// Mitsubishi GX Works2 project: 0924최신화   PLC: Q02U

PROGRAM INPUT
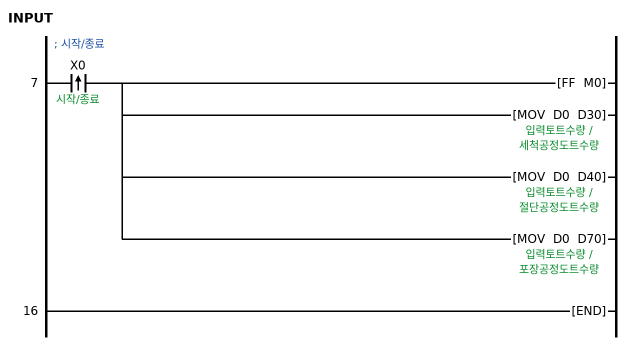
; 시작/종료
7     LDP     X0  ; 시작/종료
      FF      M0
      MOV     D0 D30  ; 입력토트수량 / 세척공정도트수량
      MOV     D0 D40  ; 절단공정도트수량
      MOV     D0 D70  ; 포장공정도트수량
16    END
END_PROGRAM

PROGRAM 세척공정
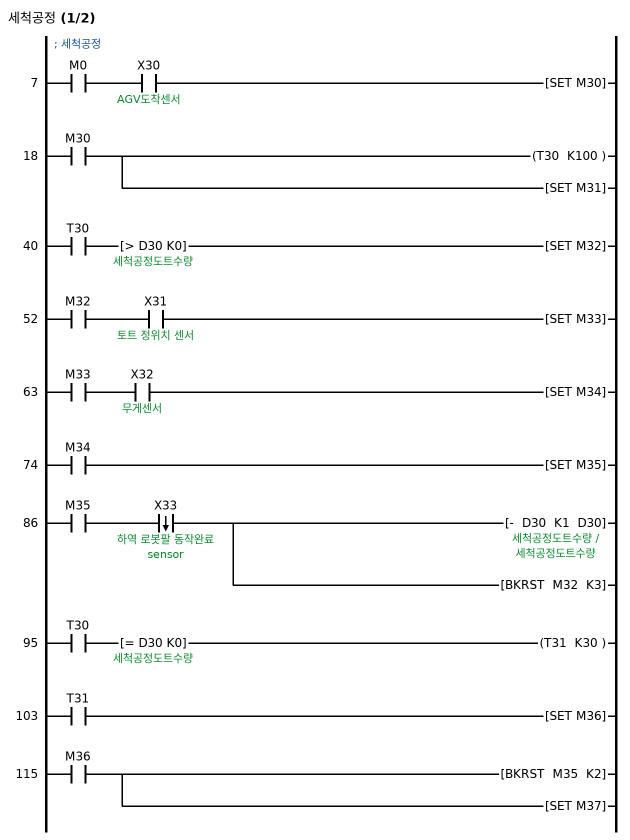
; 세척공정
7     LD      M0
      AND     X30  ; AGV도착센서
      SET     M30
        [note] 펌프모터 ON
18    LD      M30
      OUT     T30 K100
        [note] 펌핑모터 OFF
      SET     M31
        [note] SubCVY ON
40    LD      T30
      AND>    D30 K0  ; 세척공정도트수량
      SET     M32
        [note] 토트 발생
52    LD      M32
      AND     X31  ; 토트 정위치 센서
      SET     M33
        [note] MainCVY ON
63    LD      M33
      AND     X32  ; 무게센서
      SET     M34
        [note] MAinCVY OFF
74    LD      M34
      SET     M35
        [note] 하역 로봇팔 ON
86    LD      M35
      ANDF    X33  ; 하역 로봇팔 동작완료 sensor
      -       D30 K1 D30
      BKRST   M32 K3
95    LD      T30
      AND=    D30 K0  ; 세척공정도트수량
      OUT     T31 K30
103   LD      T31
      SET     M36
        [note] 하역 로봇팔 OFF
115   LD      M36
      BKRST   M35 K2
      SET     M37
        [note] AGV 다음 공정 이동, SubCVY OFF
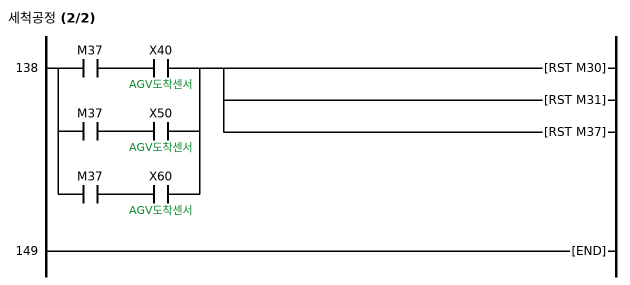
138   LD      M37
      AND     X40  ; AGV도착센서
      LD      M37
      AND     X50  ; AGV도착센서
      ORB
      LD      M37
      AND     X60  ; AGV도착센서
      ORB
      RST     M30
      RST     M31
      RST     M37
149   END
END_PROGRAM

PROGRAM 열풍건조
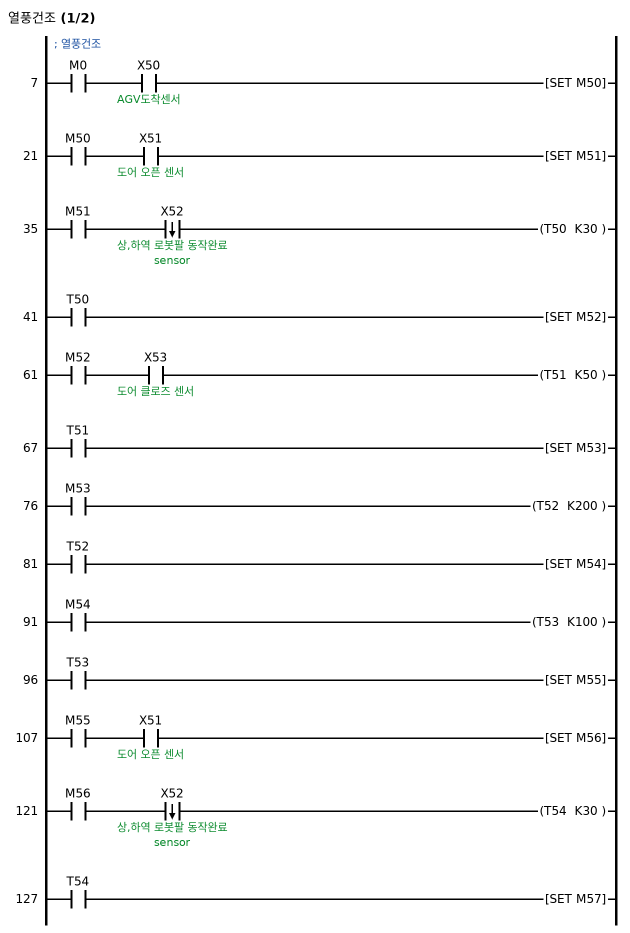
; 열풍건조
7     LD      M0
      AND     X50  ; AGV도착센서
      SET     M50
        [note] 도어 오픈모터(정)
21    LD      M50
      AND     X51  ; 도어 오픈 센서
      SET     M51
        [note] 상역 로봇 팔동작
35    LD      M51
      ANDF    X52  ; 상,하역 로봇팔 동작완료 sensor
      OUT     T50 K30
41    LD      T50
      SET     M52
        [note] 도어 클로즈모터(정), 로봇팔 OFF
61    LD      M52
      AND     X53  ; 도어 클로즈 센서
      OUT     T51 K50
67    LD      T51
      SET     M53
        [note] 건조기 ON
76    LD      M53
      OUT     T52 K200
81    LD      T52
      SET     M54
        [note] 건조기 OFF
91    LD      M54
      OUT     T53 K100
96    LD      T53
      SET     M55
        [note] 도어 오픈CYL
107   LD      M55
      AND     X51  ; 도어 오픈 센서
      SET     M56
        [note] 하역 로봇팔 동작
121   LD      M56
      ANDF    X52  ; 상,하역 로봇팔 동작완료 sensor
      OUT     T54 K30
127   LD      T54
      SET     M57
        [note] 도어 클로즈CYL, 로봇팔 OFF
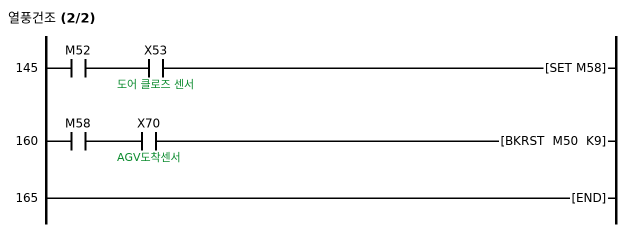
145   LD      M52
      AND     X53  ; 도어 클로즈 센서
      SET     M58
        [note] AGV 다음 공정 이동
160   LD      M58
      AND     X70  ; AGV도착센서
      BKRST   M50 K9
165   END
END_PROGRAM

PROGRAM OUTPUT
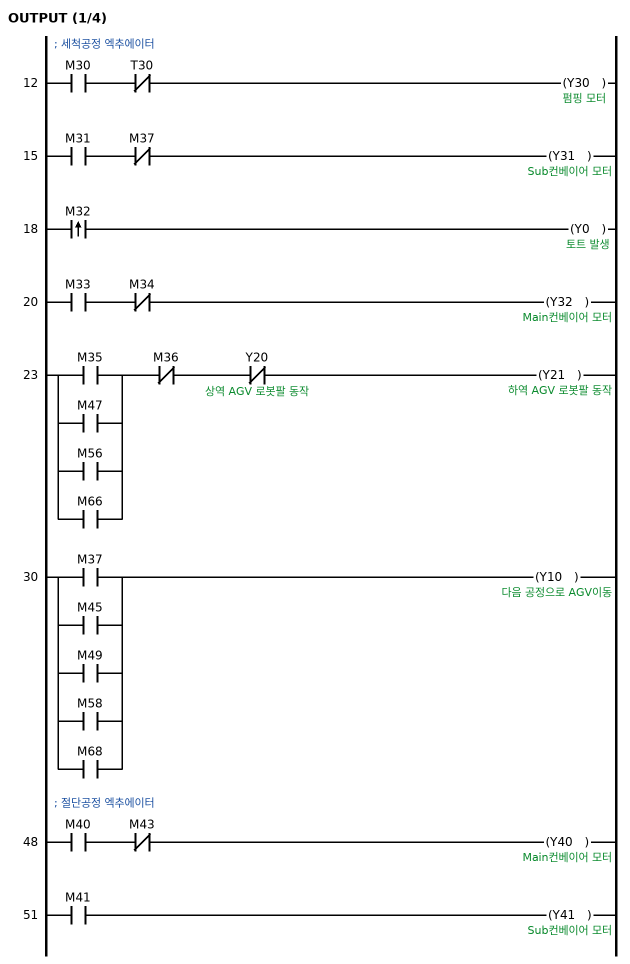
; 세척공정 엑추에이터
12    LD      M30
      ANI     T30
      OUT     Y30  ; 펌핑 모터
15    LD      M31
      ANI     M37
      OUT     Y31  ; Sub컨베이어 모터
18    LDP     M32
      OUT     Y0  ; 토트 발생
20    LD      M33
      ANI     M34
      OUT     Y32  ; Main컨베이어 모터
23    LD      M35
      OR      M47
      OR      M56
      OR      M66
      ANI     M36
      ANI     Y20  ; 상역 AGV 로봇팔 동작
      OUT     Y21  ; 하역 AGV 로봇팔 동작
30    LD      M37
      OR      M45
      OR      M49
      OR      M58
      OR      M68
      OUT     Y10  ; 다음 공정으로 AGV이동
; 절단공정 엑추에이터
48    LD      M40
      ANI     M43
      OUT     Y40  ; Main컨베이어 모터
51    LD      M41
      OUT     Y41  ; Sub컨베이어 모터
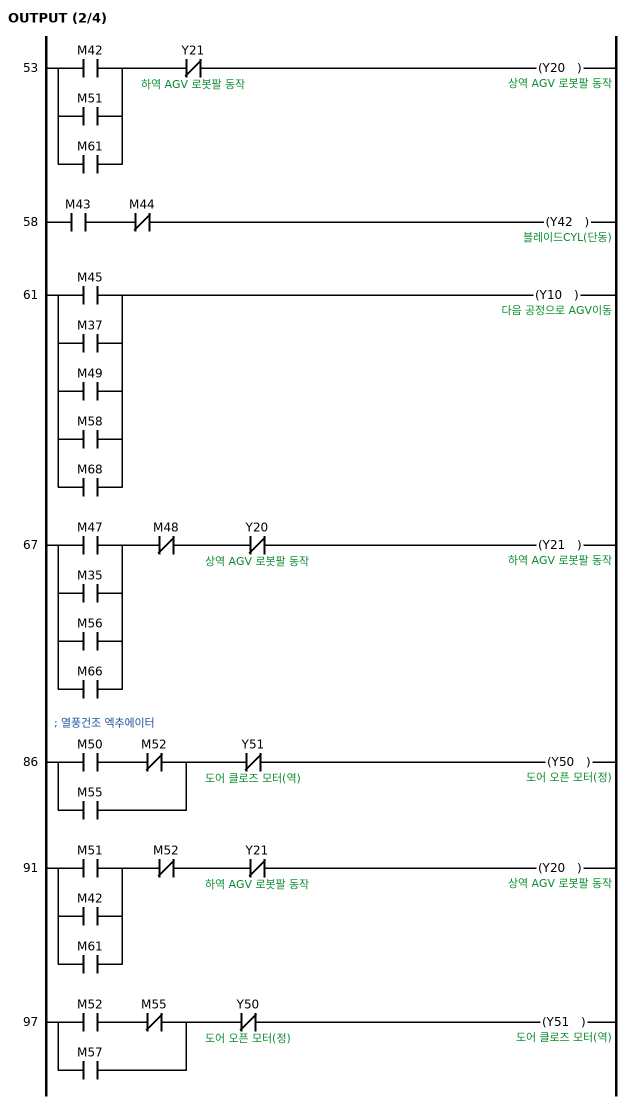
53    LD      M42
      OR      M51
      OR      M61
      ANI     Y21  ; 하역 AGV 로봇팔 동작
      OUT     Y20  ; 상역 AGV 로봇팔 동작
58    LD      M43
      ANI     M44
      OUT     Y42  ; 블레이드CYL(단동)
61    LD      M45
      OR      M37
      OR      M49
      OR      M58
      OR      M68
      OUT     Y10  ; 다음 공정으로 AGV이동
67    LD      M47
      OR      M35
      OR      M56
      OR      M66
      ANI     M48
      ANI     Y20  ; 상역 AGV 로봇팔 동작
      OUT     Y21  ; 하역 AGV 로봇팔 동작
; 열풍건조 엑추에이터
86    LD      M50
      ANI     M52
      OR      M55
      ANI     Y51  ; 도어 클로즈 모터(역)
      OUT     Y50  ; 도어 오픈 모터(정)
91    LD      M51
      OR      M42
      OR      M61
      ANI     M52
      ANI     Y21  ; 하역 AGV 로봇팔 동작
      OUT     Y20  ; 상역 AGV 로봇팔 동작
97    LD      M52
      ANI     M55
      OR      M57
      ANI     Y50  ; 도어 오픈 모터(정)
      OUT     Y51  ; 도어 클로즈 모터(역)
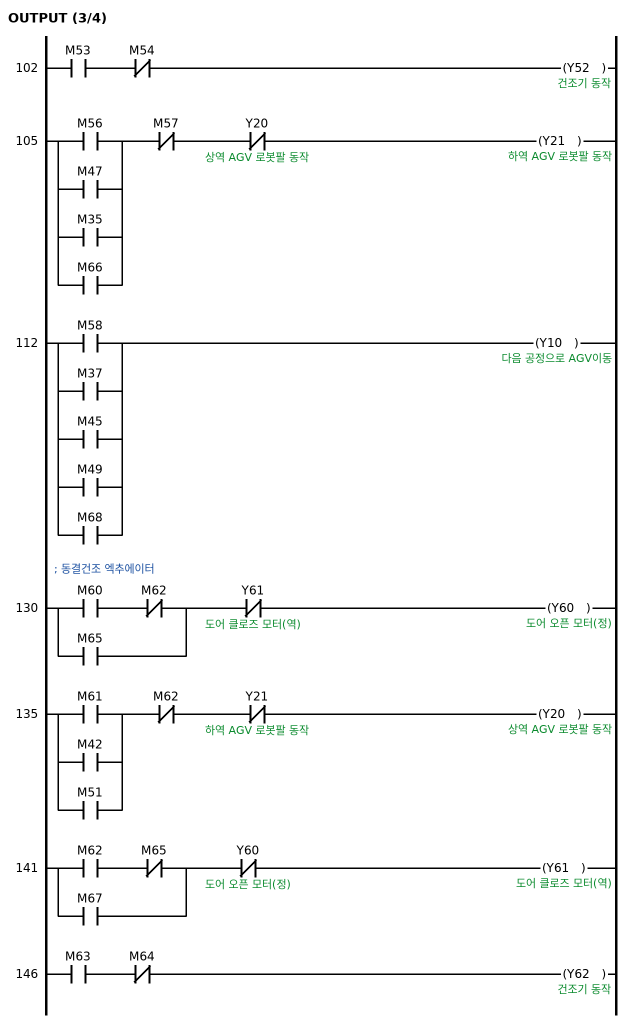
102   LD      M53
      ANI     M54
      OUT     Y52  ; 건조기 동작
105   LD      M56
      OR      M47
      OR      M35
      OR      M66
      ANI     M57
      ANI     Y20  ; 상역 AGV 로봇팔 동작
      OUT     Y21  ; 하역 AGV 로봇팔 동작
112   LD      M58
      OR      M37
      OR      M45
      OR      M49
      OR      M68
      OUT     Y10  ; 다음 공정으로 AGV이동
; 동결건조 엑추에이터
130   LD      M60
      ANI     M62
      OR      M65
      ANI     Y61  ; 도어 클로즈 모터(역)
      OUT     Y60  ; 도어 오픈 모터(정)
135   LD      M61
      OR      M42
      OR      M51
      ANI     M62
      ANI     Y21  ; 하역 AGV 로봇팔 동작
      OUT     Y20  ; 상역 AGV 로봇팔 동작
141   LD      M62
      ANI     M65
      OR      M67
      ANI     Y60  ; 도어 오픈 모터(정)
      OUT     Y61  ; 도어 클로즈 모터(역)
146   LD      M63
      ANI     M64
      OUT     Y62  ; 건조기 동작
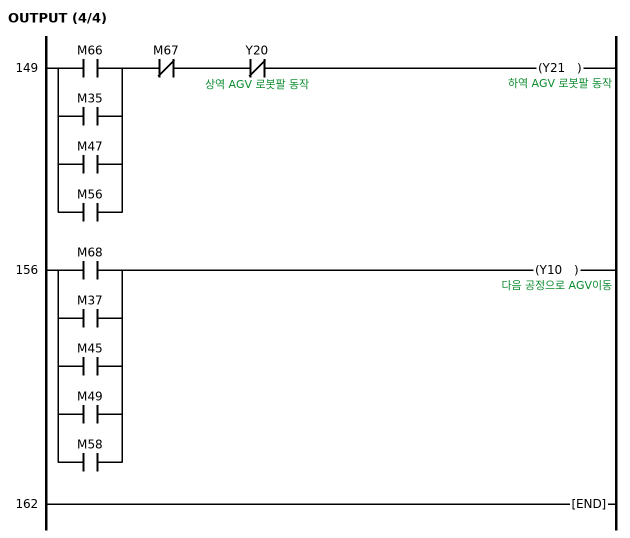
149   LD      M66
      OR      M35
      OR      M47
      OR      M56
      ANI     M67
      ANI     Y20  ; 상역 AGV 로봇팔 동작
      OUT     Y21  ; 하역 AGV 로봇팔 동작
156   LD      M68
      OR      M37
      OR      M45
      OR      M49
      OR      M58
      OUT     Y10  ; 다음 공정으로 AGV이동
162   END
END_PROGRAM

PROGRAM 동결건조
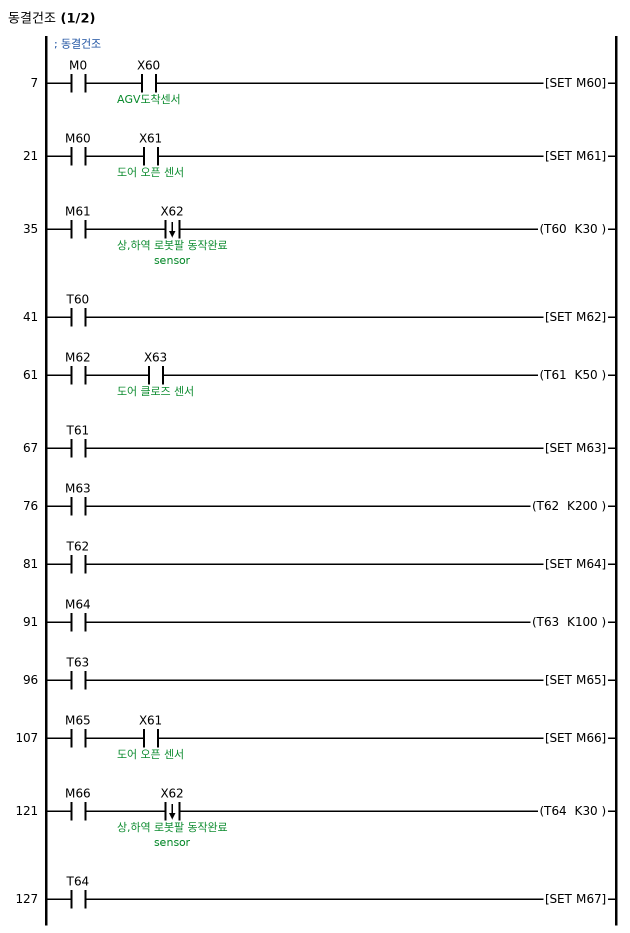
; 동결건조
7     LD      M0
      AND     X60  ; AGV도착센서
      SET     M60
        [note] 도어 오픈모터(정)
21    LD      M60
      AND     X61  ; 도어 오픈 센서
      SET     M61
        [note] 상역 로봇 팔동작
35    LD      M61
      ANDF    X62  ; 상,하역 로봇팔 동작완료 sensor
      OUT     T60 K30
41    LD      T60
      SET     M62
        [note] 도어 클로즈모터(정),로봇팔 OFF
61    LD      M62
      AND     X63  ; 도어 클로즈 센서
      OUT     T61 K50
67    LD      T61
      SET     M63
        [note] 건조기 ON
76    LD      M63
      OUT     T62 K200
81    LD      T62
      SET     M64
        [note] 건조기 OFF
91    LD      M64
      OUT     T63 K100
96    LD      T63
      SET     M65
        [note] 도어 오픈CYL
107   LD      M65
      AND     X61  ; 도어 오픈 센서
      SET     M66
        [note] 하역 로봇팔 동작
121   LD      M66
      ANDF    X62  ; 상,하역 로봇팔 동작완료 sensor
      OUT     T64 K30
127   LD      T64
      SET     M67
        [note] 도어 클로즈CYL, 로봇팔 OFF
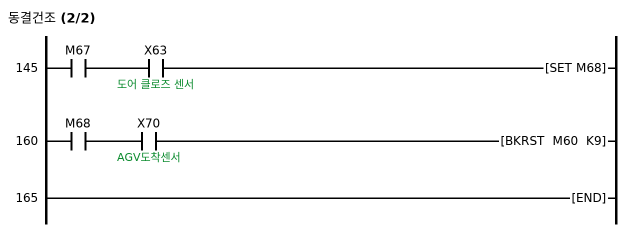
145   LD      M67
      AND     X63  ; 도어 클로즈 센서
      SET     M68
        [note] AGV 다음 공정 이동
160   LD      M68
      AND     X70  ; AGV도착센서
      BKRST   M60 K9
165   END
END_PROGRAM

PROGRAM 절단공정
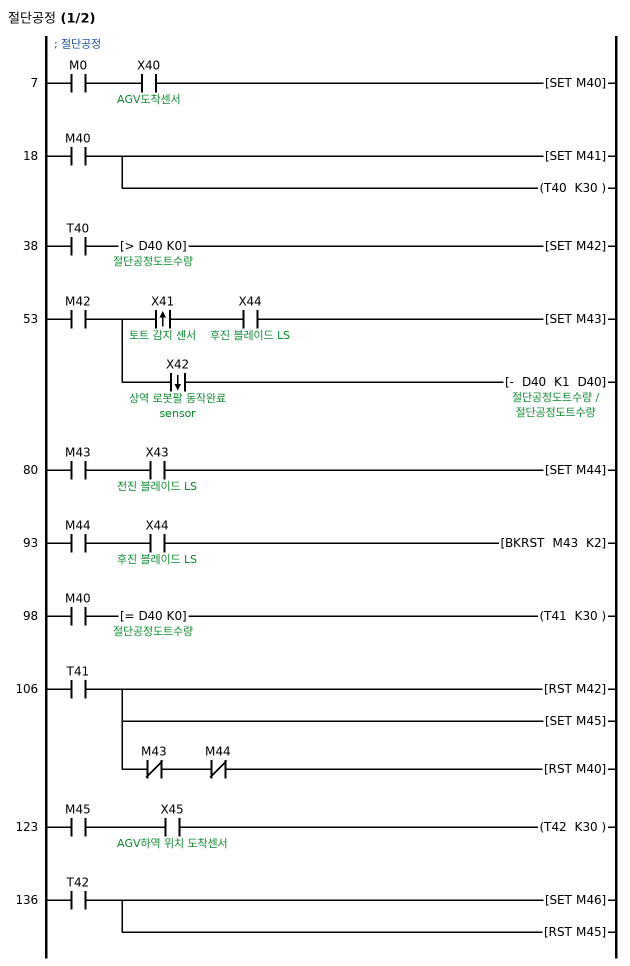
; 절단공정
7     LD      M0
      AND     X40  ; AGV도착센서
      SET     M40
        [note] MainCVY ON
18    LD      M40
      SET     M41
        [note] SubCVY ON
      OUT     T40 K30
        [note] 상역 여유
38    LD      T40
      AND>    D40 K0  ; 절단공정도트수량
      SET     M42
        [note] 상역 로봇팔 ON
53    LD      M42
      MPS
      ANDP    X41  ; 토트 감지 센서
      AND     X44  ; 후진 블레이드 LS
      SET     M43
        [note] MainCVY OFF, 블레이드CYL ON
      MPP
      ANDF    X42  ; 상역 로봇팔 동작완료 sensor
      -       D40 K1 D40
80    LD      M43
      AND     X43  ; 전진 블레이드 LS
      SET     M44
        [note] 블레이드CYL OFF
93    LD      M44
      AND     X44  ; 후진 블레이드 LS
      BKRST   M43 K2
98    LD      M40
      AND=    D40 K0  ; 절단공정도트수량
      OUT     T41 K30
106   LD      T41
      RST     M42
      SET     M45
        [note] AGV하역 위치 이동
      ANI     M43
      ANI     M44
      RST     M40
123   LD      M45
      AND     X45  ; AGV하역 위치 도착센서
      OUT     T42 K30
        [note] 하역 여유
136   LD      T42
      SET     M46
      RST     M45
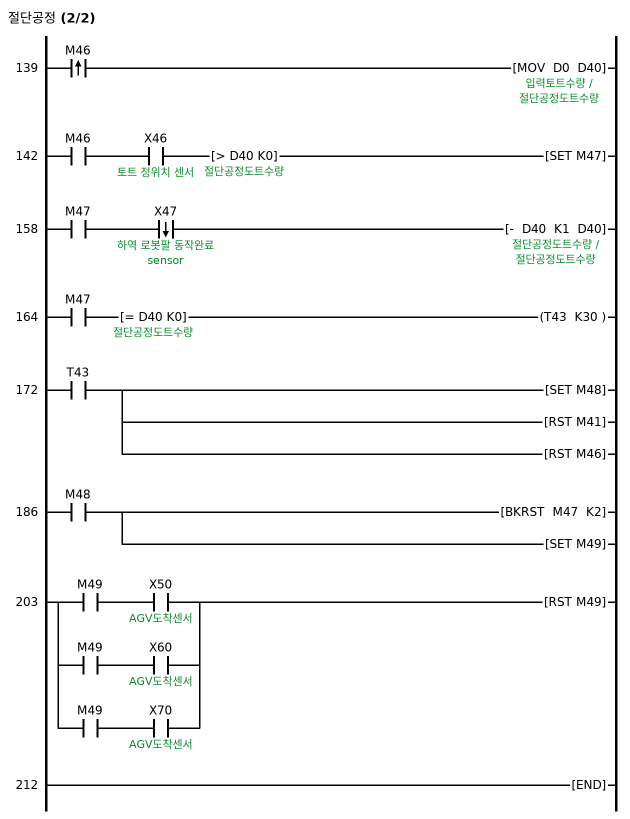
139   LDP     M46
      MOV     D0 D40  ; 입력토트수량
142   LD      M46
      AND     X46  ; 토트 정위치 센서
      AND>    D40 K0  ; 절단공정도트수량
      SET     M47
        [note] 하역 로봇팔 ON
158   LD      M47
      ANDF    X47  ; 하역 로봇팔 동작완료 sensor
      -       D40 K1 D40
164   LD      M47
      AND=    D40 K0  ; 절단공정도트수량
      OUT     T43 K30
172   LD      T43
      SET     M48
        [note] 하역 로봇팔 OFF
      RST     M41
      RST     M46
186   LD      M48
      BKRST   M47 K2
      SET     M49
        [note] AGV 다음 공정 이동
203   LD      M49
      AND     X50  ; AGV도착센서
      LD      M49
      AND     X60  ; AGV도착센서
      ORB
      LD      M49
      AND     X70  ; AGV도착센서
      ORB
      RST     M49
212   END
END_PROGRAM

// device comments not shown above
X12  ; 토틀 감지 센서
X20  ; 로봇팔 동작완료 근접sensor
D50  ; 열풍건조공정도트수량
D60  ; 동결건조공정도트수량
